// TIA Portal V18 export
DATA_BLOCK "MotorData"   // DB3120
{ S7_Optimized_Access := 'FALSE' }
// stored: AutoNumber false
   VAR
      Ton : Array[0..50] of TON_TIME;
      P { S7_SetPoint := 'True'} : Array[0..50] of Bool;
      "Time" : Array[0..50] of Time;
   END_VAR
BEGIN
   "Time"[0..50] := T#60s;
END_DATA_BLOCK
